(* CODESYS project CaseRefrigeration.project

Project tree, tasks and I/O mapping:
  PLC_AC500_V3 : PM5012-R-ETH, ABB Automation Products GmbH, order no. 1SAP122700R0072, version 3.4.1.0
    application Application
      task Task (cyclic, interval t#10ms, priority 15, watchdog t#20ms x 1) calls PLC_PRG
      CheckConfigurationObject
      program PLC_PRG [ST]
      global variables GVL
    OnBoard_IO : 6DI/4DO-R, ABB Automation Products GmbH, version 3.4.1.0
        unmapped channels: Fast inputs DI0-DI3, Fast inputs DI4-DI5, Relay outputs NO0-NO3
    Interfaces : Interfaces, ABB Automation Products GmbH, version 3.4.1.0
      OptionSlot_1
      Ethernet : Ethernet, ABB Automation Products GmbH, version 3.4.1.0
        ETH1 : IP Settings, ABB Automation Products GmbH, version 3.4.1.0
          NetConfig : NetConfig, ABB Automation Products GmbH, version 3.4.0.0
        Protocols : Client Protocols, ABB Automation Products GmbH, version 3.4.1.0
*)

// PLC_AC500_V3/Application/GVL
{attribute 'qualified_only'}
VAR_GLOBAL
// Global Variables for Case Automation

AiroffSensor:REAL;
AirOnSensor:REAL;
DefrostSensor:REAL;
DefrostHeater:REAL;
DoorSensor:BOOL;
DefrostOn:BOOL;
CompressorOn:BOOL;
DewPointSensor:REAL;
HumiditySensor:REAL;
AmbientSensor:REAL;
AirOnFan:REAL;

END_VAR

// PLC_AC500_V3/Application/PLC_PRG
PROGRAM PLC_PRG
VAR
	
END_VAR

END_PROGRAM
